TYPE TRunStatus :
	(
		RS_WaitRequest,
		RS_ProcessRequest1,
		RS_ProcessRequest2,
		RS_NotRunning
	);
END_TYPE

(* stored: Version 1.1.0.1, ProductVersion 3.1.4022.12
   DUT TRunStatus: Id {2e72993d-03e6-4ac8-8a62-a0f5b3207657} *)
